// Mitsubishi GX Works2 project: 수위풀이   PLC: Q02/Q02H

PROGRAM MAIN
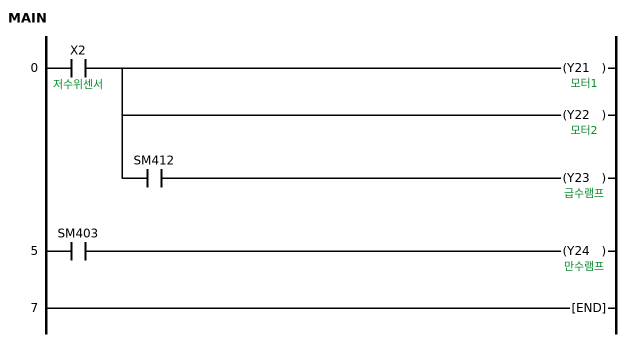
0     LD      X2  ; 저수위센서
      OUT     Y21  ; 모터1
      OUT     Y22  ; 모터2
      AND     SM412
      OUT     Y23  ; 급수램프
5     LD      SM403
      OUT     Y24  ; 만수램프
7     END
END_PROGRAM

// device comments not shown above
X0  ; 고수위센서
X1  ; 중수위센서
M0  ; 보조0
M1  ; 보조1
M2  ; 보조2
M3  ; 보조3
